TYPE ST_ToolData :
STRUCT
	// Tool Data (Value 2)
	ToolData: ARRAY [1..37] OF BYTE;
END_STRUCT
END_TYPE

(* stored: Version 1.1.0.1, ProductVersion 3.1.4020.12
   DUT ST_ToolData: Id {a33ec890-6dd0-49ca-ba62-99accd2172f6} *)
